TYPE testData :
UNION
    buffer : ARRAY[0..9999] OF BYTE;
    bufferString : STRING[9998]; 
END_UNION
END_TYPE

(* stored: Version 1.1.0.1, ProductVersion 3.1.4020.12
   DUT testData: Id {ff293035-59a6-46f3-bf60-ee1d94a35fbc} *)
